{attribute 'enable_dynamic_creation'}
FUNCTION_BLOCK INTERNAL FB_TxtLogger IMPLEMENTS ILogger
VAR_INPUT
END_VAR
VAR_OUTPUT
END_VAR
VAR
END_VAR

METHOD PUBLIC Write : STRING
VAR_INPUT
	sMsg : STRING;
END_VAR
Write := CONCAT('TxtLogger: ', sMsg);
END_METHOD

END_FUNCTION_BLOCK

(* stored: Version 1.1.0.1, ProductVersion 3.1.4024.12
   POU FB_TxtLogger: Id {b64d3bd5-8a36-4960-8962-cec44a61b481}, SpecialFunc None
   Method Write: Id {228a2bba-1d4f-4698-a869-5e758d44a93a} *)
